// TIA Portal V19 export
FUNCTION "A0303_TraslazioneStrato_CALL" : Void   // FC146, LAD
// stored: SetENOAutomatically false
BEGIN

REGION Network 1: <<< LATO TESTA >>>
END_REGION

REGION Network 2: DataIn - Asse Orizzontale
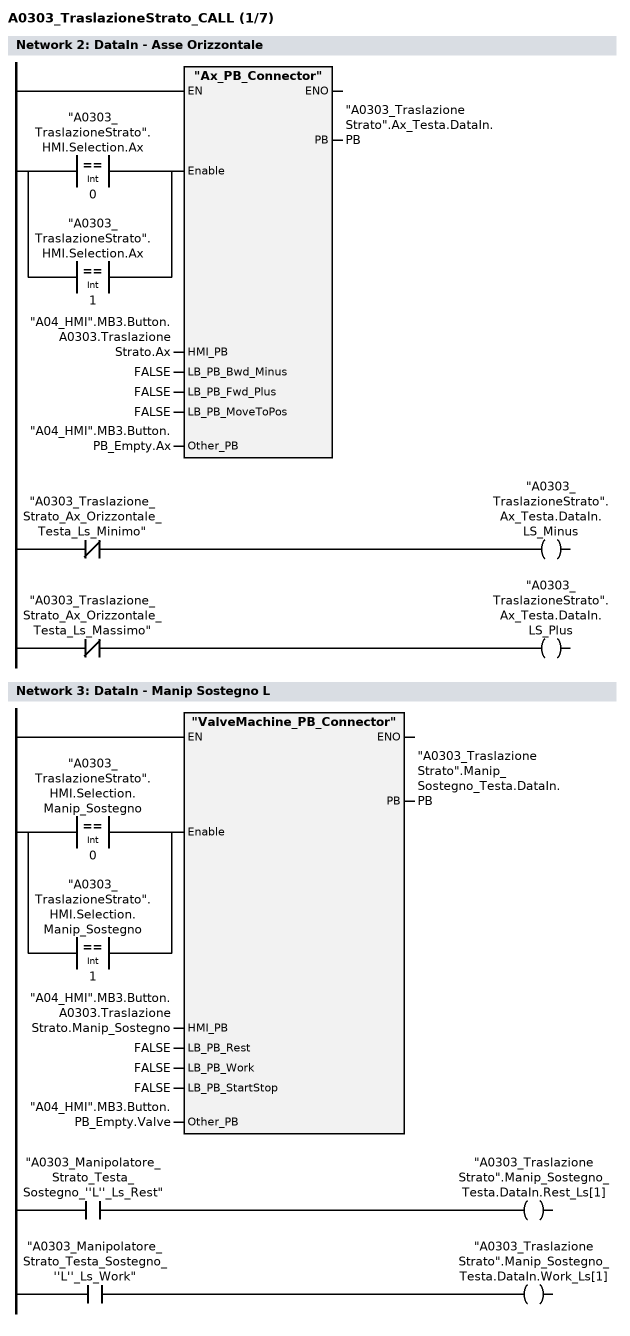
   RUNG wire#powerrail
      "Ax_PB_Connector"(Enable := wire#w1, HMI_PB := "A04_HMI".MB3.Button.A0303.TraslazioneStrato.Ax, LB_PB_Bwd_Minus := FALSE, LB_PB_Fwd_Plus := FALSE, LB_PB_MoveToPos := FALSE, Other_PB := "A04_HMI".MB3.Button.PB_Empty.Ax, PB => "A0303_TraslazioneStrato".Ax_Testa.DataIn.PB)
   END_RUNG
   RUNG wire#powerrail
      { S7_Templates := "SrcType := Int" } EQ_Contact(in1 := "A0303_TraslazioneStrato".HMI.Selection.Ax, in2 := 0)
   END_RUNG wire#w1
   RUNG wire#powerrail
      { S7_Templates := "SrcType := Int" } EQ_Contact(in1 := "A0303_TraslazioneStrato".HMI.Selection.Ax, in2 := 1)
   END_RUNG wire#w1
   RUNG wire#powerrail
      I_Contact( "A0303_Traslazione_Strato_Ax_Orizzontale_Testa_Ls_Minimo" )
      Coil( "A0303_TraslazioneStrato".Ax_Testa.DataIn.LS_Minus )
   END_RUNG
   RUNG wire#powerrail
      I_Contact( "A0303_Traslazione_Strato_Ax_Orizzontale_Testa_Ls_Massimo" )
      Coil( "A0303_TraslazioneStrato".Ax_Testa.DataIn.LS_Plus )
   END_RUNG
   // the same network as SCL:
   "Ax_PB_Connector"(Enable := ("A0303_TraslazioneStrato".HMI.Selection.Ax = 0) OR ("A0303_TraslazioneStrato".HMI.Selection.Ax = 1),
                     HMI_PB := "A04_HMI".MB3.Button.A0303.TraslazioneStrato.Ax,
                     LB_PB_Bwd_Minus := FALSE,
                     LB_PB_Fwd_Plus := FALSE,
                     LB_PB_MoveToPos := FALSE,
                     Other_PB := "A04_HMI".MB3.Button.PB_Empty.Ax,
                     PB => "A0303_TraslazioneStrato".Ax_Testa.DataIn.PB);
   "A0303_TraslazioneStrato".Ax_Testa.DataIn.LS_Minus := NOT "A0303_Traslazione_Strato_Ax_Orizzontale_Testa_Ls_Minimo";
   "A0303_TraslazioneStrato".Ax_Testa.DataIn.LS_Plus := NOT "A0303_Traslazione_Strato_Ax_Orizzontale_Testa_Ls_Massimo";
END_REGION

REGION Network 3: DataIn - Manip Sostegno L
   RUNG wire#powerrail
      "ValveMachine_PB_Connector"(Enable := wire#w1, HMI_PB := "A04_HMI".MB3.Button.A0303.TraslazioneStrato.Manip_Sostegno, LB_PB_Rest := FALSE, LB_PB_Work := FALSE, LB_PB_StartStop := FALSE, Other_PB := "A04_HMI".MB3.Button.PB_Empty.Valve, PB => "A0303_TraslazioneStrato".Manip_Sostegno_Testa.DataIn.PB)
   END_RUNG
   RUNG wire#powerrail
      { S7_Templates := "SrcType := Int" } EQ_Contact(in1 := "A0303_TraslazioneStrato".HMI.Selection.Manip_Sostegno, in2 := 0)
   END_RUNG wire#w1
   RUNG wire#powerrail
      { S7_Templates := "SrcType := Int" } EQ_Contact(in1 := "A0303_TraslazioneStrato".HMI.Selection.Manip_Sostegno, in2 := 1)
   END_RUNG wire#w1
   RUNG wire#powerrail
      Contact( "A0303_Manipolatore_Strato_Testa_Sostegno_''L''_Ls_Rest" )
      Coil( "A0303_TraslazioneStrato".Manip_Sostegno_Testa.DataIn.Rest_Ls[1] )
   END_RUNG
   RUNG wire#powerrail
      Contact( "A0303_Manipolatore_Strato_Testa_Sostegno_''L''_Ls_Work" )
      Coil( "A0303_TraslazioneStrato".Manip_Sostegno_Testa.DataIn.Work_Ls[1] )
   END_RUNG
   // the same network as SCL:
   "ValveMachine_PB_Connector"(Enable := ("A0303_TraslazioneStrato".HMI.Selection.Manip_Sostegno = 0) OR ("A0303_TraslazioneStrato".HMI.Selection.Manip_Sostegno = 1),
                           HMI_PB := "A04_HMI".MB3.Button.A0303.TraslazioneStrato.Manip_Sostegno,
                           LB_PB_Rest := FALSE,
                           LB_PB_Work := FALSE,
                           LB_PB_StartStop := FALSE,
                           Other_PB := "A04_HMI".MB3.Button.PB_Empty.Valve,
                           PB => "A0303_TraslazioneStrato".Manip_Sostegno_Testa.DataIn.PB);
   "A0303_TraslazioneStrato".Manip_Sostegno_Testa.DataIn.Rest_Ls[1] := "A0303_Manipolatore_Strato_Testa_Sostegno_''L''_Ls_Rest";
   "A0303_TraslazioneStrato".Manip_Sostegno_Testa.DataIn.Work_Ls[1] := "A0303_Manipolatore_Strato_Testa_Sostegno_''L''_Ls_Work";
END_REGION

REGION Network 4: DataIn - Manip Pareggiatore
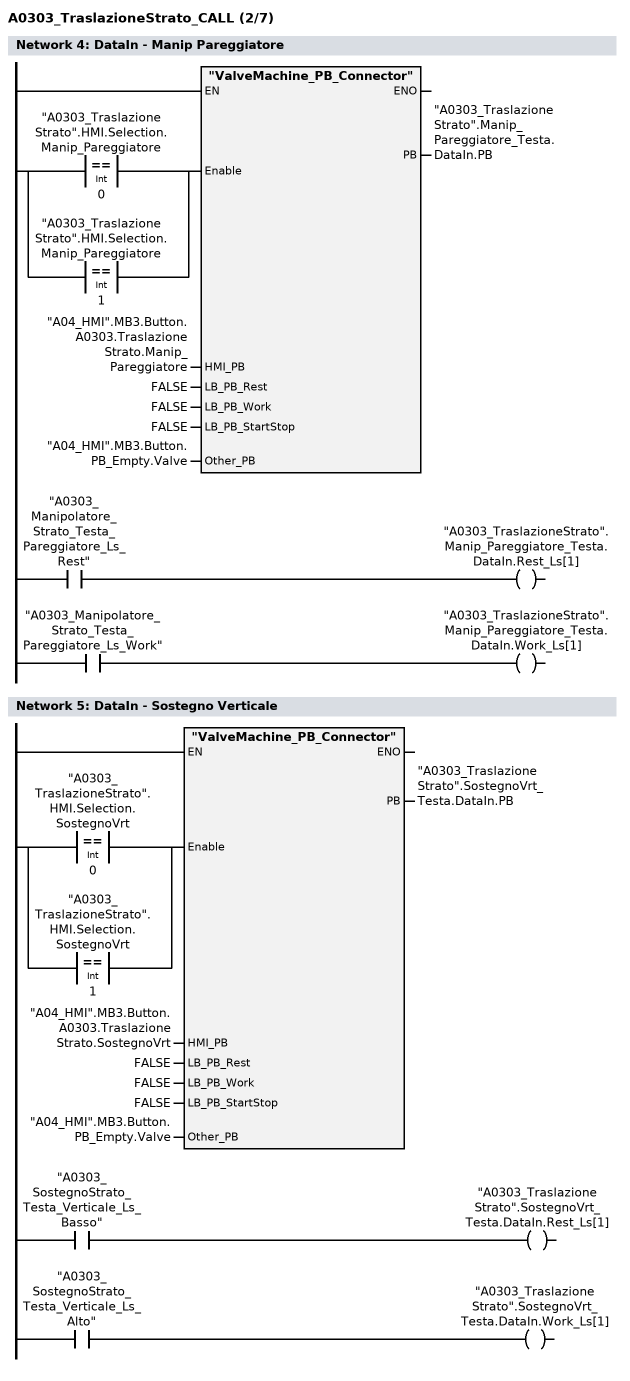
   RUNG wire#powerrail
      "ValveMachine_PB_Connector"(Enable := wire#w1, HMI_PB := "A04_HMI".MB3.Button.A0303.TraslazioneStrato.Manip_Pareggiatore, LB_PB_Rest := FALSE, LB_PB_Work := FALSE, LB_PB_StartStop := FALSE, Other_PB := "A04_HMI".MB3.Button.PB_Empty.Valve, PB => "A0303_TraslazioneStrato".Manip_Pareggiatore_Testa.DataIn.PB)
   END_RUNG
   RUNG wire#powerrail
      { S7_Templates := "SrcType := Int" } EQ_Contact(in1 := "A0303_TraslazioneStrato".HMI.Selection.Manip_Pareggiatore, in2 := 0)
   END_RUNG wire#w1
   RUNG wire#powerrail
      { S7_Templates := "SrcType := Int" } EQ_Contact(in1 := "A0303_TraslazioneStrato".HMI.Selection.Manip_Pareggiatore, in2 := 1)
   END_RUNG wire#w1
   RUNG wire#powerrail
      Contact( "A0303_Manipolatore_Strato_Testa_Pareggiatore_Ls_Rest" )
      Coil( "A0303_TraslazioneStrato".Manip_Pareggiatore_Testa.DataIn.Rest_Ls[1] )
   END_RUNG
   RUNG wire#powerrail
      Contact( "A0303_Manipolatore_Strato_Testa_Pareggiatore_Ls_Work" )
      Coil( "A0303_TraslazioneStrato".Manip_Pareggiatore_Testa.DataIn.Work_Ls[1] )
   END_RUNG
   // the same network as SCL:
   "ValveMachine_PB_Connector"(Enable := ("A0303_TraslazioneStrato".HMI.Selection.Manip_Pareggiatore = 0) OR ("A0303_TraslazioneStrato".HMI.Selection.Manip_Pareggiatore = 1),
                           HMI_PB := "A04_HMI".MB3.Button.A0303.TraslazioneStrato.Manip_Pareggiatore,
                           LB_PB_Rest := FALSE,
                           LB_PB_Work := FALSE,
                           LB_PB_StartStop := FALSE,
                           Other_PB := "A04_HMI".MB3.Button.PB_Empty.Valve,
                           PB => "A0303_TraslazioneStrato".Manip_Pareggiatore_Testa.DataIn.PB);
   "A0303_TraslazioneStrato".Manip_Pareggiatore_Testa.DataIn.Rest_Ls[1] := "A0303_Manipolatore_Strato_Testa_Pareggiatore_Ls_Rest";
   "A0303_TraslazioneStrato".Manip_Pareggiatore_Testa.DataIn.Work_Ls[1] := "A0303_Manipolatore_Strato_Testa_Pareggiatore_Ls_Work";
END_REGION

REGION Network 5: DataIn - Sostegno Verticale
   RUNG wire#powerrail
      "ValveMachine_PB_Connector"(Enable := wire#w1, HMI_PB := "A04_HMI".MB3.Button.A0303.TraslazioneStrato.SostegnoVrt, LB_PB_Rest := FALSE, LB_PB_Work := FALSE, LB_PB_StartStop := FALSE, Other_PB := "A04_HMI".MB3.Button.PB_Empty.Valve, PB => "A0303_TraslazioneStrato".SostegnoVrt_Testa.DataIn.PB)
   END_RUNG
   RUNG wire#powerrail
      { S7_Templates := "SrcType := Int" } EQ_Contact(in1 := "A0303_TraslazioneStrato".HMI.Selection.SostegnoVrt, in2 := 0)
   END_RUNG wire#w1
   RUNG wire#powerrail
      { S7_Templates := "SrcType := Int" } EQ_Contact(in1 := "A0303_TraslazioneStrato".HMI.Selection.SostegnoVrt, in2 := 1)
   END_RUNG wire#w1
   RUNG wire#powerrail
      Contact( "A0303_SostegnoStrato_Testa_Verticale_Ls_Basso" )
      Coil( "A0303_TraslazioneStrato".SostegnoVrt_Testa.DataIn.Rest_Ls[1] )
   END_RUNG
   RUNG wire#powerrail
      Contact( "A0303_SostegnoStrato_Testa_Verticale_Ls_Alto" )
      Coil( "A0303_TraslazioneStrato".SostegnoVrt_Testa.DataIn.Work_Ls[1] )
   END_RUNG
   // the same network as SCL:
   "ValveMachine_PB_Connector"(Enable := ("A0303_TraslazioneStrato".HMI.Selection.SostegnoVrt = 0) OR ("A0303_TraslazioneStrato".HMI.Selection.SostegnoVrt = 1),
                           HMI_PB := "A04_HMI".MB3.Button.A0303.TraslazioneStrato.SostegnoVrt,
                           LB_PB_Rest := FALSE,
                           LB_PB_Work := FALSE,
                           LB_PB_StartStop := FALSE,
                           Other_PB := "A04_HMI".MB3.Button.PB_Empty.Valve,
                           PB => "A0303_TraslazioneStrato".SostegnoVrt_Testa.DataIn.PB);
   "A0303_TraslazioneStrato".SostegnoVrt_Testa.DataIn.Rest_Ls[1] := "A0303_SostegnoStrato_Testa_Verticale_Ls_Basso";
   "A0303_TraslazioneStrato".SostegnoVrt_Testa.DataIn.Work_Ls[1] := "A0303_SostegnoStrato_Testa_Verticale_Ls_Alto";
END_REGION

REGION Network 6: DataIn -Analog Sensor
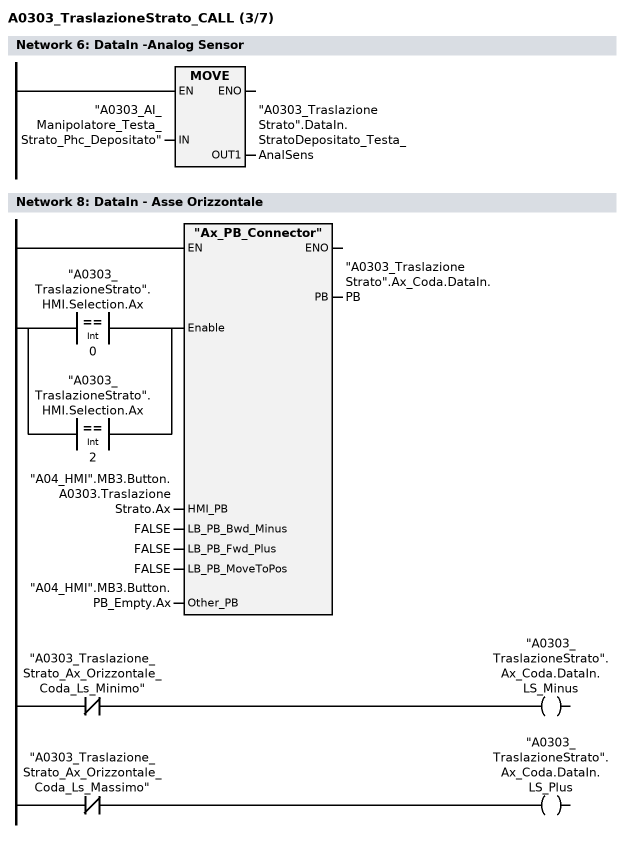
   RUNG wire#powerrail
      Move(in := "A0303_AI_Manipolatore_Testa_Strato_Phc_Depositato", out1 => "A0303_TraslazioneStrato".DataIn.StratoDepositato_Testa_AnalSens)
   END_RUNG
   // the same network as SCL:
   "A0303_TraslazioneStrato".DataIn.StratoDepositato_Testa_AnalSens := "A0303_AI_Manipolatore_Testa_Strato_Phc_Depositato";
END_REGION

REGION Network 7: <<< LATO CODA >>>
END_REGION

REGION Network 8: DataIn - Asse Orizzontale
   RUNG wire#powerrail
      "Ax_PB_Connector"(Enable := wire#w1, HMI_PB := "A04_HMI".MB3.Button.A0303.TraslazioneStrato.Ax, LB_PB_Bwd_Minus := FALSE, LB_PB_Fwd_Plus := FALSE, LB_PB_MoveToPos := FALSE, Other_PB := "A04_HMI".MB3.Button.PB_Empty.Ax, PB => "A0303_TraslazioneStrato".Ax_Coda.DataIn.PB)
   END_RUNG
   RUNG wire#powerrail
      { S7_Templates := "SrcType := Int" } EQ_Contact(in1 := "A0303_TraslazioneStrato".HMI.Selection.Ax, in2 := 0)
   END_RUNG wire#w1
   RUNG wire#powerrail
      { S7_Templates := "SrcType := Int" } EQ_Contact(in1 := "A0303_TraslazioneStrato".HMI.Selection.Ax, in2 := 2)
   END_RUNG wire#w1
   RUNG wire#powerrail
      I_Contact( "A0303_Traslazione_Strato_Ax_Orizzontale_Coda_Ls_Minimo" )
      Coil( "A0303_TraslazioneStrato".Ax_Coda.DataIn.LS_Minus )
   END_RUNG
   RUNG wire#powerrail
      I_Contact( "A0303_Traslazione_Strato_Ax_Orizzontale_Coda_Ls_Massimo" )
      Coil( "A0303_TraslazioneStrato".Ax_Coda.DataIn.LS_Plus )
   END_RUNG
   // the same network as SCL:
   "Ax_PB_Connector"(Enable := ("A0303_TraslazioneStrato".HMI.Selection.Ax = 0) OR ("A0303_TraslazioneStrato".HMI.Selection.Ax = 2),
                     HMI_PB := "A04_HMI".MB3.Button.A0303.TraslazioneStrato.Ax,
                     LB_PB_Bwd_Minus := FALSE,
                     LB_PB_Fwd_Plus := FALSE,
                     LB_PB_MoveToPos := FALSE,
                     Other_PB := "A04_HMI".MB3.Button.PB_Empty.Ax,
                     PB => "A0303_TraslazioneStrato".Ax_Coda.DataIn.PB);
   "A0303_TraslazioneStrato".Ax_Coda.DataIn.LS_Minus := NOT "A0303_Traslazione_Strato_Ax_Orizzontale_Coda_Ls_Minimo";
   "A0303_TraslazioneStrato".Ax_Coda.DataIn.LS_Plus := NOT "A0303_Traslazione_Strato_Ax_Orizzontale_Coda_Ls_Massimo";
END_REGION

REGION Network 9: DataIn - Manip Sostegno L
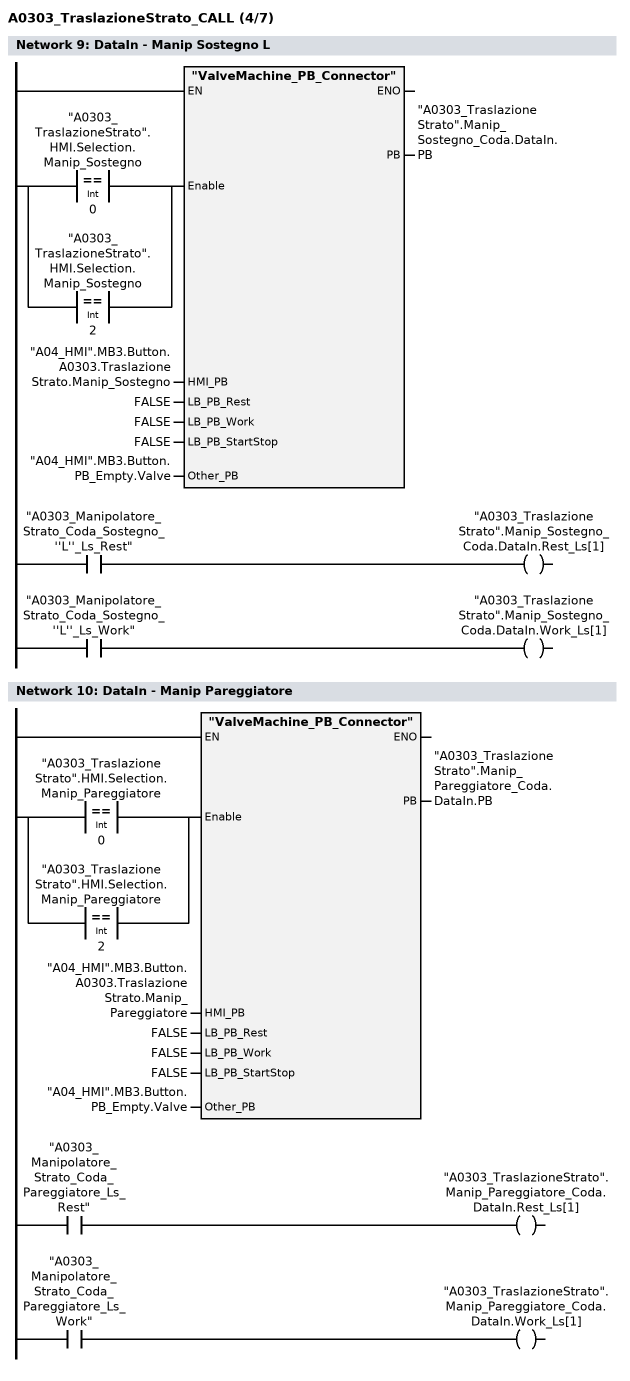
   RUNG wire#powerrail
      "ValveMachine_PB_Connector"(Enable := wire#w1, HMI_PB := "A04_HMI".MB3.Button.A0303.TraslazioneStrato.Manip_Sostegno, LB_PB_Rest := FALSE, LB_PB_Work := FALSE, LB_PB_StartStop := FALSE, Other_PB := "A04_HMI".MB3.Button.PB_Empty.Valve, PB => "A0303_TraslazioneStrato".Manip_Sostegno_Coda.DataIn.PB)
   END_RUNG
   RUNG wire#powerrail
      { S7_Templates := "SrcType := Int" } EQ_Contact(in1 := "A0303_TraslazioneStrato".HMI.Selection.Manip_Sostegno, in2 := 0)
   END_RUNG wire#w1
   RUNG wire#powerrail
      { S7_Templates := "SrcType := Int" } EQ_Contact(in1 := "A0303_TraslazioneStrato".HMI.Selection.Manip_Sostegno, in2 := 2)
   END_RUNG wire#w1
   RUNG wire#powerrail
      Contact( "A0303_Manipolatore_Strato_Coda_Sostegno_''L''_Ls_Rest" )
      Coil( "A0303_TraslazioneStrato".Manip_Sostegno_Coda.DataIn.Rest_Ls[1] )
   END_RUNG
   RUNG wire#powerrail
      Contact( "A0303_Manipolatore_Strato_Coda_Sostegno_''L''_Ls_Work" )
      Coil( "A0303_TraslazioneStrato".Manip_Sostegno_Coda.DataIn.Work_Ls[1] )
   END_RUNG
   // the same network as SCL:
   "ValveMachine_PB_Connector"(Enable := ("A0303_TraslazioneStrato".HMI.Selection.Manip_Sostegno = 0) OR ("A0303_TraslazioneStrato".HMI.Selection.Manip_Sostegno = 2),
                           HMI_PB := "A04_HMI".MB3.Button.A0303.TraslazioneStrato.Manip_Sostegno,
                           LB_PB_Rest := FALSE,
                           LB_PB_Work := FALSE,
                           LB_PB_StartStop := FALSE,
                           Other_PB := "A04_HMI".MB3.Button.PB_Empty.Valve,
                           PB => "A0303_TraslazioneStrato".Manip_Sostegno_Coda.DataIn.PB);
   "A0303_TraslazioneStrato".Manip_Sostegno_Coda.DataIn.Rest_Ls[1] := "A0303_Manipolatore_Strato_Coda_Sostegno_''L''_Ls_Rest";
   "A0303_TraslazioneStrato".Manip_Sostegno_Coda.DataIn.Work_Ls[1] := "A0303_Manipolatore_Strato_Coda_Sostegno_''L''_Ls_Work";
END_REGION

REGION Network 10: DataIn - Manip Pareggiatore
   RUNG wire#powerrail
      "ValveMachine_PB_Connector"(Enable := wire#w1, HMI_PB := "A04_HMI".MB3.Button.A0303.TraslazioneStrato.Manip_Pareggiatore, LB_PB_Rest := FALSE, LB_PB_Work := FALSE, LB_PB_StartStop := FALSE, Other_PB := "A04_HMI".MB3.Button.PB_Empty.Valve, PB => "A0303_TraslazioneStrato".Manip_Pareggiatore_Coda.DataIn.PB)
   END_RUNG
   RUNG wire#powerrail
      { S7_Templates := "SrcType := Int" } EQ_Contact(in1 := "A0303_TraslazioneStrato".HMI.Selection.Manip_Pareggiatore, in2 := 0)
   END_RUNG wire#w1
   RUNG wire#powerrail
      { S7_Templates := "SrcType := Int" } EQ_Contact(in1 := "A0303_TraslazioneStrato".HMI.Selection.Manip_Pareggiatore, in2 := 2)
   END_RUNG wire#w1
   RUNG wire#powerrail
      Contact( "A0303_Manipolatore_Strato_Coda_Pareggiatore_Ls_Rest" )
      Coil( "A0303_TraslazioneStrato".Manip_Pareggiatore_Coda.DataIn.Rest_Ls[1] )
   END_RUNG
   RUNG wire#powerrail
      Contact( "A0303_Manipolatore_Strato_Coda_Pareggiatore_Ls_Work" )
      Coil( "A0303_TraslazioneStrato".Manip_Pareggiatore_Coda.DataIn.Work_Ls[1] )
   END_RUNG
   // the same network as SCL:
   "ValveMachine_PB_Connector"(Enable := ("A0303_TraslazioneStrato".HMI.Selection.Manip_Pareggiatore = 0) OR ("A0303_TraslazioneStrato".HMI.Selection.Manip_Pareggiatore = 2),
                           HMI_PB := "A04_HMI".MB3.Button.A0303.TraslazioneStrato.Manip_Pareggiatore,
                           LB_PB_Rest := FALSE,
                           LB_PB_Work := FALSE,
                           LB_PB_StartStop := FALSE,
                           Other_PB := "A04_HMI".MB3.Button.PB_Empty.Valve,
                           PB => "A0303_TraslazioneStrato".Manip_Pareggiatore_Coda.DataIn.PB);
   "A0303_TraslazioneStrato".Manip_Pareggiatore_Coda.DataIn.Rest_Ls[1] := "A0303_Manipolatore_Strato_Coda_Pareggiatore_Ls_Rest";
   "A0303_TraslazioneStrato".Manip_Pareggiatore_Coda.DataIn.Work_Ls[1] := "A0303_Manipolatore_Strato_Coda_Pareggiatore_Ls_Work";
END_REGION

REGION Network 11: DataIn - Sostegno Verticale
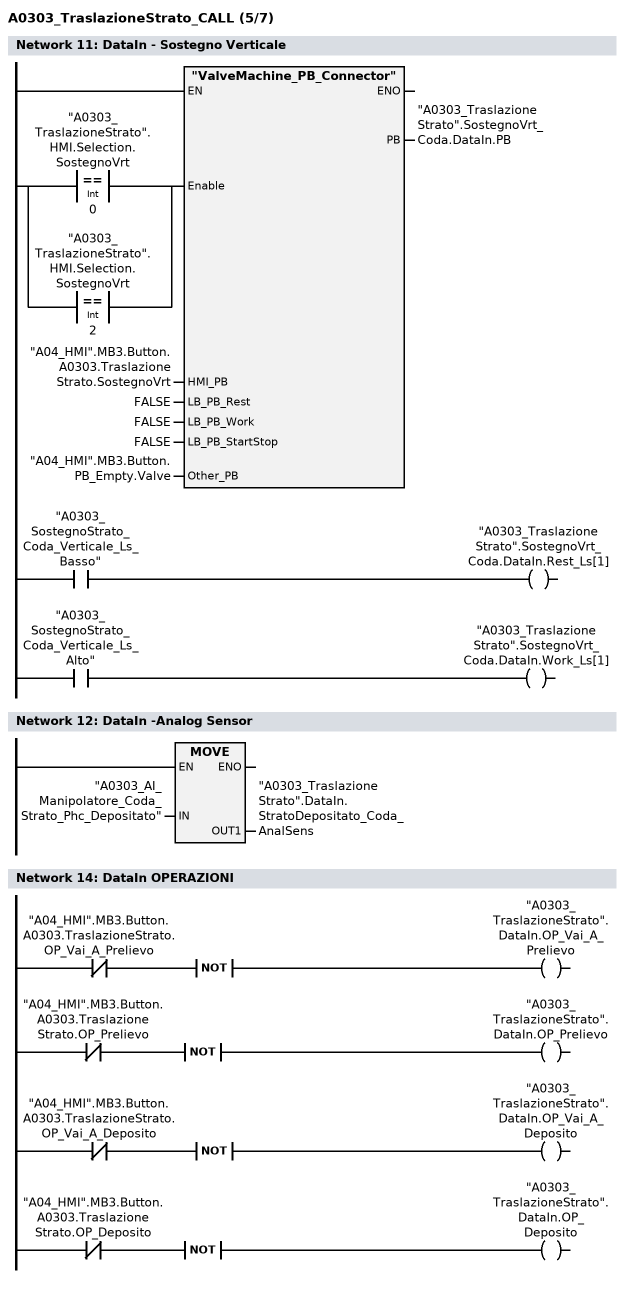
   RUNG wire#powerrail
      "ValveMachine_PB_Connector"(Enable := wire#w1, HMI_PB := "A04_HMI".MB3.Button.A0303.TraslazioneStrato.SostegnoVrt, LB_PB_Rest := FALSE, LB_PB_Work := FALSE, LB_PB_StartStop := FALSE, Other_PB := "A04_HMI".MB3.Button.PB_Empty.Valve, PB => "A0303_TraslazioneStrato".SostegnoVrt_Coda.DataIn.PB)
   END_RUNG
   RUNG wire#powerrail
      { S7_Templates := "SrcType := Int" } EQ_Contact(in1 := "A0303_TraslazioneStrato".HMI.Selection.SostegnoVrt, in2 := 0)
   END_RUNG wire#w1
   RUNG wire#powerrail
      { S7_Templates := "SrcType := Int" } EQ_Contact(in1 := "A0303_TraslazioneStrato".HMI.Selection.SostegnoVrt, in2 := 2)
   END_RUNG wire#w1
   RUNG wire#powerrail
      Contact( "A0303_SostegnoStrato_Coda_Verticale_Ls_Basso" )
      Coil( "A0303_TraslazioneStrato".SostegnoVrt_Coda.DataIn.Rest_Ls[1] )
   END_RUNG
   RUNG wire#powerrail
      Contact( "A0303_SostegnoStrato_Coda_Verticale_Ls_Alto" )
      Coil( "A0303_TraslazioneStrato".SostegnoVrt_Coda.DataIn.Work_Ls[1] )
   END_RUNG
   // the same network as SCL:
   "ValveMachine_PB_Connector"(Enable := ("A0303_TraslazioneStrato".HMI.Selection.SostegnoVrt = 0) OR ("A0303_TraslazioneStrato".HMI.Selection.SostegnoVrt = 2),
                           HMI_PB := "A04_HMI".MB3.Button.A0303.TraslazioneStrato.SostegnoVrt,
                           LB_PB_Rest := FALSE,
                           LB_PB_Work := FALSE,
                           LB_PB_StartStop := FALSE,
                           Other_PB := "A04_HMI".MB3.Button.PB_Empty.Valve,
                           PB => "A0303_TraslazioneStrato".SostegnoVrt_Coda.DataIn.PB);
   "A0303_TraslazioneStrato".SostegnoVrt_Coda.DataIn.Rest_Ls[1] := "A0303_SostegnoStrato_Coda_Verticale_Ls_Basso";
   "A0303_TraslazioneStrato".SostegnoVrt_Coda.DataIn.Work_Ls[1] := "A0303_SostegnoStrato_Coda_Verticale_Ls_Alto";
END_REGION

REGION Network 12: DataIn -Analog Sensor
   RUNG wire#powerrail
      Move(in := "A0303_AI_Manipolatore_Coda_Strato_Phc_Depositato", out1 => "A0303_TraslazioneStrato".DataIn.StratoDepositato_Coda_AnalSens)
   END_RUNG
   // the same network as SCL:
   "A0303_TraslazioneStrato".DataIn.StratoDepositato_Coda_AnalSens := "A0303_AI_Manipolatore_Coda_Strato_Phc_Depositato";
END_REGION

REGION Network 14: DataIn OPERAZIONI
   RUNG wire#powerrail
      I_Contact( "A04_HMI".MB3.Button.A0303.TraslazioneStrato.OP_Vai_A_Prelievo )
      Not()
      Coil( "A0303_TraslazioneStrato".DataIn.OP_Vai_A_Prelievo )
   END_RUNG
   RUNG wire#powerrail
      I_Contact( "A04_HMI".MB3.Button.A0303.TraslazioneStrato.OP_Prelievo )
      Not()
      Coil( "A0303_TraslazioneStrato".DataIn.OP_Prelievo )
   END_RUNG
   RUNG wire#powerrail
      I_Contact( "A04_HMI".MB3.Button.A0303.TraslazioneStrato.OP_Vai_A_Deposito )
      Not()
      Coil( "A0303_TraslazioneStrato".DataIn.OP_Vai_A_Deposito )
   END_RUNG
   RUNG wire#powerrail
      I_Contact( "A04_HMI".MB3.Button.A0303.TraslazioneStrato.OP_Deposito )
      Not()
      Coil( "A0303_TraslazioneStrato".DataIn.OP_Deposito )
   END_RUNG
   // the same network as SCL:
   "A0303_TraslazioneStrato".DataIn.OP_Vai_A_Prelievo := NOT (NOT "A04_HMI".MB3.Button.A0303.TraslazioneStrato.OP_Vai_A_Prelievo);
   "A0303_TraslazioneStrato".DataIn.OP_Prelievo := NOT (NOT "A04_HMI".MB3.Button.A0303.TraslazioneStrato.OP_Prelievo);
   "A0303_TraslazioneStrato".DataIn.OP_Vai_A_Deposito := NOT (NOT "A04_HMI".MB3.Button.A0303.TraslazioneStrato.OP_Vai_A_Deposito);
   "A0303_TraslazioneStrato".DataIn.OP_Deposito := NOT (NOT "A04_HMI".MB3.Button.A0303.TraslazioneStrato.OP_Deposito);
END_REGION

REGION Network 16: CIn
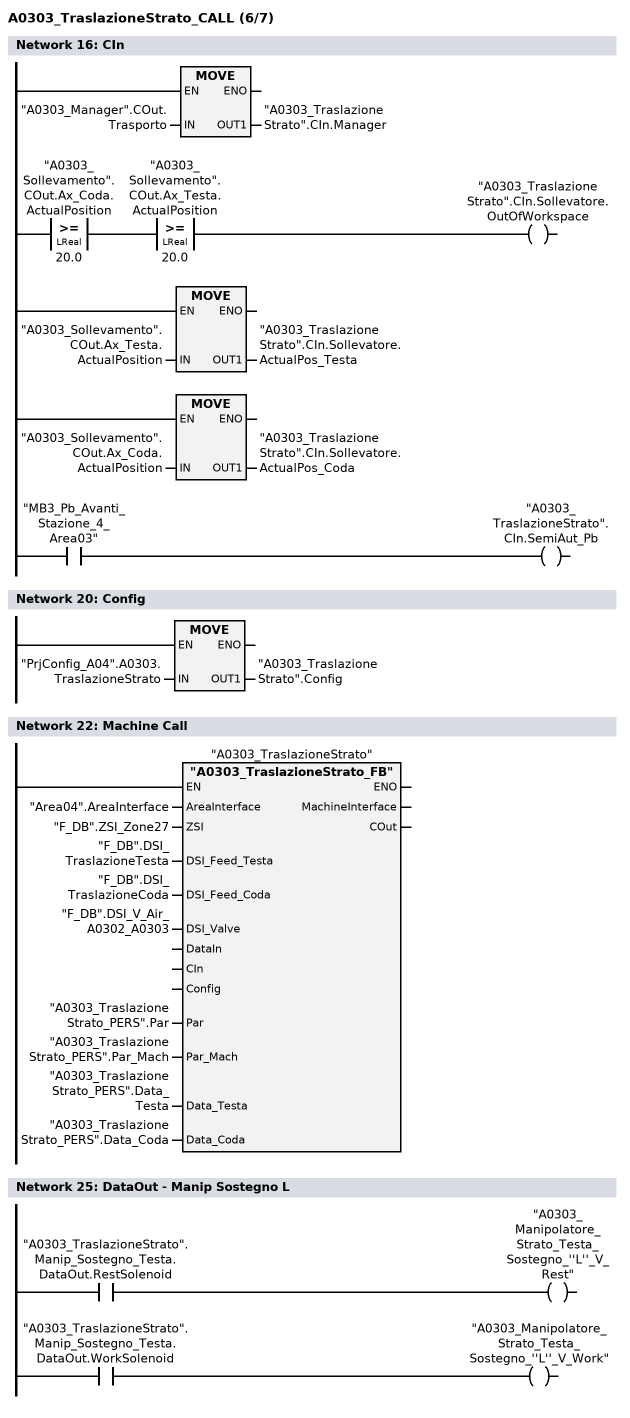
   RUNG wire#powerrail
      Move(in := "A0303_Manager".COut.Trasporto, out1 => "A0303_TraslazioneStrato".CIn.Manager)
   END_RUNG
   RUNG wire#powerrail
      { S7_Templates := "SrcType := LReal" } GE_Contact(in1 := "A0303_Sollevamento".COut.Ax_Coda.ActualPosition, in2 := 20.0)
      { S7_Templates := "SrcType := LReal" } GE_Contact(in1 := "A0303_Sollevamento".COut.Ax_Testa.ActualPosition, in2 := 20.0)
      Coil( "A0303_TraslazioneStrato".CIn.Sollevatore.OutOfWorkspace )
   END_RUNG
   RUNG wire#powerrail
      Move(in := "A0303_Sollevamento".COut.Ax_Testa.ActualPosition, out1 => "A0303_TraslazioneStrato".CIn.Sollevatore.ActualPos_Testa)
   END_RUNG
   RUNG wire#powerrail
      Move(in := "A0303_Sollevamento".COut.Ax_Coda.ActualPosition, out1 => "A0303_TraslazioneStrato".CIn.Sollevatore.ActualPos_Coda)
   END_RUNG
   RUNG wire#powerrail
      Contact( "MB3_Pb_Avanti_Stazione_4_Area03" )
      Coil( "A0303_TraslazioneStrato".CIn.SemiAut_Pb )
   END_RUNG
   // the same network as SCL:
   "A0303_TraslazioneStrato".CIn.Manager := "A0303_Manager".COut.Trasporto;
   "A0303_TraslazioneStrato".CIn.Sollevatore.OutOfWorkspace := ("A0303_Sollevamento".COut.Ax_Coda.ActualPosition >= 20.0) AND ("A0303_Sollevamento".COut.Ax_Testa.ActualPosition >= 20.0);
   "A0303_TraslazioneStrato".CIn.Sollevatore.ActualPos_Testa := "A0303_Sollevamento".COut.Ax_Testa.ActualPosition;
   "A0303_TraslazioneStrato".CIn.Sollevatore.ActualPos_Coda := "A0303_Sollevamento".COut.Ax_Coda.ActualPosition;
   "A0303_TraslazioneStrato".CIn.SemiAut_Pb := "MB3_Pb_Avanti_Stazione_4_Area03";
END_REGION

REGION Network 17: >
END_REGION

REGION Network 18 (SCL): Drive
   "A0303_TraslazioneStrato".Ax_Testa.Drive.Infeed_ON := "Areas_ITF".AG.Infeed_Running;
   "A0303_TraslazioneStrato".Ax_Testa.Drive.AccessPoint := "HW_Const_Values".CU7_PN_610A1_ModuleAccessPoint;
   "A0303_TraslazioneStrato".Ax_Testa.Drive.AxisID := "CU7_ID_2_2310A1_1_2310M1";
   "A0303_TraslazioneStrato".Ax_Testa.Drive.TokenChain := "TOKENCHAIN_CU7";


   "A0303_TraslazioneStrato".Ax_Coda.Drive.Infeed_ON := "Areas_ITF".AG.Infeed_Running;
   "A0303_TraslazioneStrato".Ax_Coda.Drive.AccessPoint := "HW_Const_Values".CU7_PN_610A1_ModuleAccessPoint;
   "A0303_TraslazioneStrato".Ax_Coda.Drive.AxisID :="CU7_ID_3_2310A1_2_2330M1";
   "A0303_TraslazioneStrato".Ax_Coda.Drive.TokenChain := "TOKENCHAIN_CU7";
END_REGION

REGION Network 19 (SCL): HW
   "A0303_TraslazioneStrato".Ax_Testa.HW_ID_TEL111 := "HW_Const_Values".CU7_PN_2310A1_1_SIEMENS_telegram_111;

   "A0303_TraslazioneStrato".Ax_Coda.HW_ID_TEL111 := "HW_Const_Values".CU7_PN_2310A1_2_SIEMENS_telegram_111;
END_REGION

REGION Network 20: Config
   RUNG wire#powerrail
      Move(in := "PrjConfig_A04".A0303.TraslazioneStrato, out1 => "A0303_TraslazioneStrato".Config)
   END_RUNG
   // the same network as SCL:
   "A0303_TraslazioneStrato".Config := "PrjConfig_A04".A0303.TraslazioneStrato;
END_REGION

REGION Network 21: >
END_REGION

REGION Network 22: Machine Call
   RUNG wire#powerrail
      "A0303_TraslazioneStrato"(AreaInterface := "Area04".AreaInterface, ZSI := "F_DB".ZSI_Zone27, DSI_Feed_Testa := "F_DB".DSI_TraslazioneTesta, DSI_Feed_Coda := "F_DB".DSI_TraslazioneCoda, DSI_Valve := "F_DB".DSI_V_Air_A0302_A0303, DataIn :=, CIn :=, Config :=, Par := "A0303_TraslazioneStrato_PERS".Par, Par_Mach := "A0303_TraslazioneStrato_PERS".Par_Mach, Data_Testa := "A0303_TraslazioneStrato_PERS".Data_Testa, Data_Coda := "A0303_TraslazioneStrato_PERS".Data_Coda, MachineInterface =>, COut =>)
   END_RUNG
   // the same network as SCL:
   "A0303_TraslazioneStrato"(AreaInterface := "Area04".AreaInterface,   // "A0303_TraslazioneStrato_FB"
                           ZSI := "F_DB".ZSI_Zone27,
                           DSI_Feed_Testa := "F_DB".DSI_TraslazioneTesta,
                           DSI_Feed_Coda := "F_DB".DSI_TraslazioneCoda,
                           DSI_Valve := "F_DB".DSI_V_Air_A0302_A0303,
                           Par := "A0303_TraslazioneStrato_PERS".Par,
                           Par_Mach := "A0303_TraslazioneStrato_PERS".Par_Mach,
                           Data_Testa := "A0303_TraslazioneStrato_PERS".Data_Testa,
                           Data_Coda := "A0303_TraslazioneStrato_PERS".Data_Coda);
END_REGION

REGION Network 24: <<< LATO TESTA >>>
END_REGION

REGION Network 25: DataOut - Manip Sostegno L
   RUNG wire#powerrail
      Contact( "A0303_TraslazioneStrato".Manip_Sostegno_Testa.DataOut.RestSolenoid )
      Coil( "A0303_Manipolatore_Strato_Testa_Sostegno_''L''_V_Rest" )
   END_RUNG
   RUNG wire#powerrail
      Contact( "A0303_TraslazioneStrato".Manip_Sostegno_Testa.DataOut.WorkSolenoid )
      Coil( "A0303_Manipolatore_Strato_Testa_Sostegno_''L''_V_Work" )
   END_RUNG
   // the same network as SCL:
   "A0303_Manipolatore_Strato_Testa_Sostegno_''L''_V_Rest" := "A0303_TraslazioneStrato".Manip_Sostegno_Testa.DataOut.RestSolenoid;
   "A0303_Manipolatore_Strato_Testa_Sostegno_''L''_V_Work" := "A0303_TraslazioneStrato".Manip_Sostegno_Testa.DataOut.WorkSolenoid;
END_REGION

REGION Network 26: DataOut - Pareggiatore
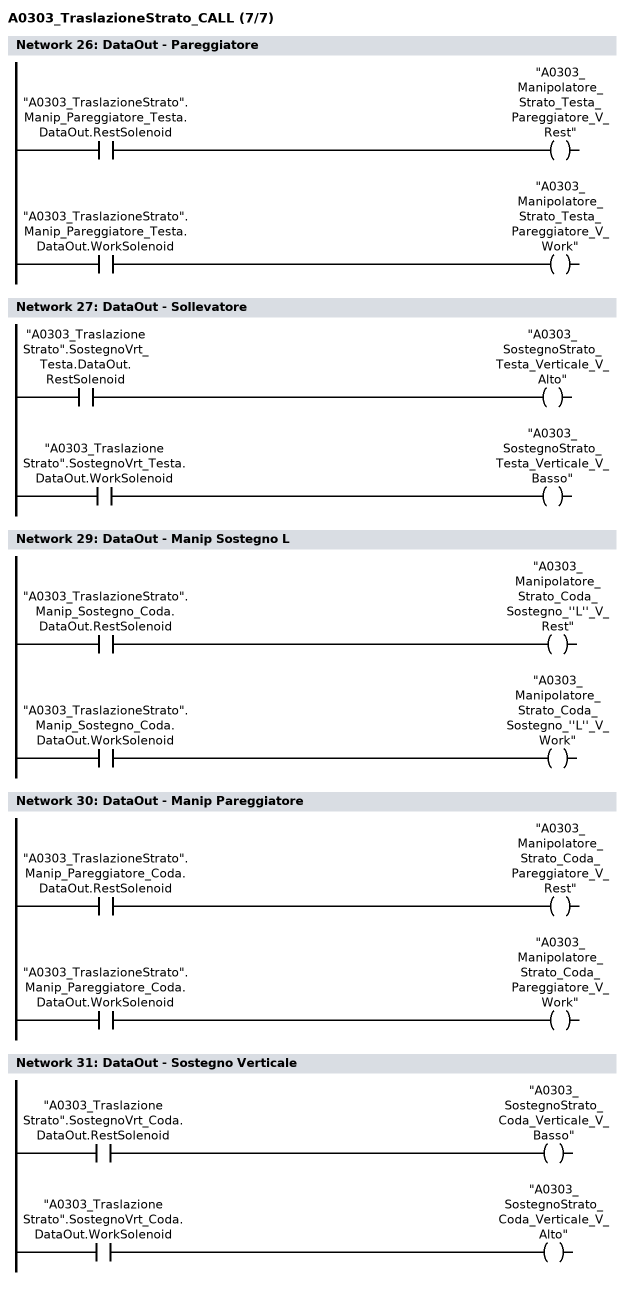
   RUNG wire#powerrail
      Contact( "A0303_TraslazioneStrato".Manip_Pareggiatore_Testa.DataOut.RestSolenoid )
      Coil( "A0303_Manipolatore_Strato_Testa_Pareggiatore_V_Rest" )
   END_RUNG
   RUNG wire#powerrail
      Contact( "A0303_TraslazioneStrato".Manip_Pareggiatore_Testa.DataOut.WorkSolenoid )
      Coil( "A0303_Manipolatore_Strato_Testa_Pareggiatore_V_Work" )
   END_RUNG
   // the same network as SCL:
   "A0303_Manipolatore_Strato_Testa_Pareggiatore_V_Rest" := "A0303_TraslazioneStrato".Manip_Pareggiatore_Testa.DataOut.RestSolenoid;
   "A0303_Manipolatore_Strato_Testa_Pareggiatore_V_Work" := "A0303_TraslazioneStrato".Manip_Pareggiatore_Testa.DataOut.WorkSolenoid;
END_REGION

REGION Network 27: DataOut - Sollevatore
   RUNG wire#powerrail
      Contact( "A0303_TraslazioneStrato".SostegnoVrt_Testa.DataOut.RestSolenoid )
      Coil( "A0303_SostegnoStrato_Testa_Verticale_V_Alto" )
   END_RUNG
   RUNG wire#powerrail
      Contact( "A0303_TraslazioneStrato".SostegnoVrt_Testa.DataOut.WorkSolenoid )
      Coil( "A0303_SostegnoStrato_Testa_Verticale_V_Basso" )
   END_RUNG
   // the same network as SCL:
   "A0303_SostegnoStrato_Testa_Verticale_V_Alto" := "A0303_TraslazioneStrato".SostegnoVrt_Testa.DataOut.RestSolenoid;
   "A0303_SostegnoStrato_Testa_Verticale_V_Basso" := "A0303_TraslazioneStrato".SostegnoVrt_Testa.DataOut.WorkSolenoid;
END_REGION

REGION Network 28: <<< LATO CODA >>>
END_REGION

REGION Network 29: DataOut - Manip Sostegno L
   RUNG wire#powerrail
      Contact( "A0303_TraslazioneStrato".Manip_Sostegno_Coda.DataOut.RestSolenoid )
      Coil( "A0303_Manipolatore_Strato_Coda_Sostegno_''L''_V_Rest" )
   END_RUNG
   RUNG wire#powerrail
      Contact( "A0303_TraslazioneStrato".Manip_Sostegno_Coda.DataOut.WorkSolenoid )
      Coil( "A0303_Manipolatore_Strato_Coda_Sostegno_''L''_V_Work" )
   END_RUNG
   // the same network as SCL:
   "A0303_Manipolatore_Strato_Coda_Sostegno_''L''_V_Rest" := "A0303_TraslazioneStrato".Manip_Sostegno_Coda.DataOut.RestSolenoid;
   "A0303_Manipolatore_Strato_Coda_Sostegno_''L''_V_Work" := "A0303_TraslazioneStrato".Manip_Sostegno_Coda.DataOut.WorkSolenoid;
END_REGION

REGION Network 30: DataOut - Manip Pareggiatore
   RUNG wire#powerrail
      Contact( "A0303_TraslazioneStrato".Manip_Pareggiatore_Coda.DataOut.RestSolenoid )
      Coil( "A0303_Manipolatore_Strato_Coda_Pareggiatore_V_Rest" )
   END_RUNG
   RUNG wire#powerrail
      Contact( "A0303_TraslazioneStrato".Manip_Pareggiatore_Coda.DataOut.WorkSolenoid )
      Coil( "A0303_Manipolatore_Strato_Coda_Pareggiatore_V_Work" )
   END_RUNG
   // the same network as SCL:
   "A0303_Manipolatore_Strato_Coda_Pareggiatore_V_Rest" := "A0303_TraslazioneStrato".Manip_Pareggiatore_Coda.DataOut.RestSolenoid;
   "A0303_Manipolatore_Strato_Coda_Pareggiatore_V_Work" := "A0303_TraslazioneStrato".Manip_Pareggiatore_Coda.DataOut.WorkSolenoid;
END_REGION

REGION Network 31: DataOut - Sostegno Verticale
   RUNG wire#powerrail
      Contact( "A0303_TraslazioneStrato".SostegnoVrt_Coda.DataOut.RestSolenoid )
      Coil( "A0303_SostegnoStrato_Coda_Verticale_V_Basso" )
   END_RUNG
   RUNG wire#powerrail
      Contact( "A0303_TraslazioneStrato".SostegnoVrt_Coda.DataOut.WorkSolenoid )
      Coil( "A0303_SostegnoStrato_Coda_Verticale_V_Alto" )
   END_RUNG
   // the same network as SCL:
   "A0303_SostegnoStrato_Coda_Verticale_V_Basso" := "A0303_TraslazioneStrato".SostegnoVrt_Coda.DataOut.RestSolenoid;
   "A0303_SostegnoStrato_Coda_Verticale_V_Alto" := "A0303_TraslazioneStrato".SostegnoVrt_Coda.DataOut.WorkSolenoid;
END_REGION
END_FUNCTION
